(* IEC 61131-3 sources: Swiity/AutomationStudio/VendingMachine, 4 files *)

(* ---- Types.typ ---- *)
(*
  Types.typ
  Vending Machine Project – User-Defined Data Types (UDT)
  IEC 61131-3 Structured Text  |  B&R Automation Studio
*)

TYPE
  (* ---------------------------------------------------------------
     State enumeration for the main vending-machine state machine
  --------------------------------------------------------------- *)
  VendingState_e : (
    STATE_IDLE         := 0,   (* Waiting for coin / card input        *)
    STATE_COIN_CHECK   := 1,   (* Validating inserted coin             *)
    STATE_SELECT       := 2,   (* Product selection active             *)
    STATE_DISPENSE     := 3,   (* Dispensing selected product          *)
    STATE_COLLECT      := 4,   (* Waiting for customer to collect      *)
    STATE_CHANGE       := 5,   (* Returning change                     *)
    STATE_ERROR        := 6,   (* Error / fault state                  *)
    STATE_MAINTENANCE  := 7    (* Maintenance / refill mode            *)
  );

  (* ---------------------------------------------------------------
     Product slot descriptor
  --------------------------------------------------------------- *)
  ProductSlot_t : STRUCT
    Name        : STRING[32];  (* Product name                         *)
    Price       : REAL;        (* Price in the local currency unit     *)
    Quantity    : UINT;        (* Remaining stock count                *)
    SlotActive  : BOOL;        (* TRUE = slot is enabled               *)
  END_STRUCT;

  (* ---------------------------------------------------------------
     Coin / payment input data
  --------------------------------------------------------------- *)
  PaymentData_t : STRUCT
    CoinInserted    : BOOL;    (* Coin-drop sensor signal              *)
    CoinValue       : REAL;    (* Value detected by coin validator     *)
    TotalCredit     : REAL;    (* Accumulated credit                   *)
    CreditAccepted  : BOOL;    (* Sufficient credit for selection      *)
  END_STRUCT;

  (* ---------------------------------------------------------------
     Sensor input bundle (mapped from Arduino via serial / I/O)
  --------------------------------------------------------------- *)
  SensorInputs_t : STRUCT
    CoinSensor       : BOOL;   (* Coin-drop detection                  *)
    ProductSensor    : BOOL;   (* Product dispensed / collected        *)
    TempSensor       : REAL;   (* Cabinet temperature (°C)             *)
    DoorSensor       : BOOL;   (* Service door open                    *)
    StockSensor      : ARRAY[0..7] OF BOOL; (* Per-slot stock presence *)
  END_STRUCT;

  (* ---------------------------------------------------------------
     Actuator output bundle (mapped to Arduino via serial / I/O)
  --------------------------------------------------------------- *)
  ActuatorOutputs_t : STRUCT
    MotorEnable      : BOOL;              (* Dispense motor enable      *)
    MotorSlot        : UINT;              (* Target slot index          *)
    ChangeMechanism  : BOOL;              (* Activate change dispenser  *)
    DisplayMsg       : STRING[64];        (* LCD / display message      *)
    StatusLED        : BOOL;              (* Status indicator LED       *)
    CoolingFan       : BOOL;              (* Cooling fan control        *)
  END_STRUCT;

END_TYPE

(* ---- Variables.var ---- *)
(*
  Variables.var
  Vending Machine Project – Global Variable Declarations
  IEC 61131-3 Structured Text  |  B&R Automation Studio
*)

VAR_GLOBAL

  (* ---------------------------------------------------------------
     State machine
  --------------------------------------------------------------- *)
  gState          : VendingState_e := STATE_IDLE;
  gPrevState      : VendingState_e := STATE_IDLE;

  (* ---------------------------------------------------------------
     Product configuration  (8 slots, indices 0..7)
  --------------------------------------------------------------- *)
  gProductSlots   : ARRAY[0..7] OF ProductSlot_t;
  gSelectedSlot   : UINT := 0;

  (* ---------------------------------------------------------------
     Payment
  --------------------------------------------------------------- *)
  gPayment        : PaymentData_t;

  (* ---------------------------------------------------------------
     I/O bundles (exchanged with Arduino via serial / fieldbus)
  --------------------------------------------------------------- *)
  gSensors        : SensorInputs_t;
  gActuators      : ActuatorOutputs_t;

  (* ---------------------------------------------------------------
     Timing
  --------------------------------------------------------------- *)
  gDispenseTimer  : TON;         (* Motor run time-out                 *)
  gCollectTimer   : TON;         (* Collect reminder time-out          *)
  gErrorTimer     : TON;         (* Error-reset delay                  *)

  (* ---------------------------------------------------------------
     Diagnostics / HMI
  --------------------------------------------------------------- *)
  gErrorCode      : UINT  := 0;
  gTotalSales     : UDINT := 0;  (* Number of successful vend cycles   *)
  gHmiMessage     : STRING[64];

END_VAR

VAR_GLOBAL CONSTANT

  (* ---------------------------------------------------------------
     Application constants
  --------------------------------------------------------------- *)
  cNumSlots           : UINT := 8;        (* Total number of product slots    *)
  cDispenseTimeMs     : TIME := T#3000ms; (* Motor run duration               *)
  cCollectTimeoutMs   : TIME := T#30000ms;(* Collect reminder after 30 s      *)
  cMinTemperature     : REAL := 2.0;      (* Min cabinet temperature (°C)     *)
  cMaxTemperature     : REAL := 10.0;     (* Max cabinet temperature (°C)     *)

END_VAR

(* ---- StateMachine.st ---- *)
(*
  StateMachine.st
  Vending Machine Project – State-Machine Logic
  IEC 61131-3 Structured Text  |  B&R Automation Studio

  Call this function block once per PLC cycle from Main.st.
*)

FUNCTION_BLOCK VendingStateMachine

VAR_INPUT
  Sensors   : SensorInputs_t;   (* Live sensor data                    *)
END_VAR

VAR_OUTPUT
  Actuators : ActuatorOutputs_t;(* Computed actuator commands          *)
  State     : VendingState_e;   (* Current state (for HMI / logging)   *)
END_VAR

VAR
  _dispenseTimer   : TON;
  _collectTimer    : TON;
  _errorTimer      : TON;
  _coinSensorPrev  : BOOL := FALSE; (* Previous coin-sensor state for edge detection *)
END_VAR

(* ---------------------------------------------------------------
   Main state-machine CASE statement
--------------------------------------------------------------- *)
CASE gState OF

  (* ---- IDLE -------------------------------------------------- *)
  STATE_IDLE:
    Actuators.DisplayMsg  := 'Insert coin';
    Actuators.StatusLED   := TRUE;
    Actuators.MotorEnable := FALSE;

    IF Sensors.CoinSensor THEN
      gState := STATE_COIN_CHECK;
    END_IF

  (* ---- COIN CHECK -------------------------------------------- *)
  STATE_COIN_CHECK:
    Actuators.DisplayMsg := 'Checking coin...';

    (* Accumulate credit on rising edge of coin sensor only *)
    IF Sensors.CoinSensor AND NOT _coinSensorPrev THEN
      gPayment.TotalCredit := gPayment.TotalCredit + gPayment.CoinValue;
    END_IF
    _coinSensorPrev := Sensors.CoinSensor;

    (* Always allow product selection once any credit exists *)
    IF gPayment.TotalCredit > 0.0 THEN
      gState := STATE_SELECT;
    END_IF

  (* ---- SELECT ------------------------------------------------ *)
  STATE_SELECT:
    Actuators.DisplayMsg := 'Select product (0-7)';

    (* Validate selection: slot must be active and affordable *)
    IF gSelectedSlot < cNumSlots
       AND gProductSlots[gSelectedSlot].SlotActive
       AND gProductSlots[gSelectedSlot].Quantity > 0
       AND gPayment.TotalCredit >= gProductSlots[gSelectedSlot].Price THEN

      gPayment.CreditAccepted := TRUE;
      gState := STATE_DISPENSE;
    END_IF

  (* ---- DISPENSE ---------------------------------------------- *)
  STATE_DISPENSE:
    Actuators.DisplayMsg      := 'Dispensing...';
    Actuators.MotorEnable     := TRUE;
    Actuators.MotorSlot       := gSelectedSlot;

    _dispenseTimer(IN := TRUE, PT := cDispenseTimeMs);

    IF _dispenseTimer.Q THEN
      _dispenseTimer(IN := FALSE);
      Actuators.MotorEnable := FALSE;

      (* Deduct price, update stock *)
      gPayment.TotalCredit                       := gPayment.TotalCredit
                                                    - gProductSlots[gSelectedSlot].Price;
      gProductSlots[gSelectedSlot].Quantity      := gProductSlots[gSelectedSlot].Quantity - 1;
      gTotalSales                                := gTotalSales + 1;

      gState := STATE_COLLECT;
    END_IF

  (* ---- COLLECT ----------------------------------------------- *)
  STATE_COLLECT:
    Actuators.DisplayMsg := 'Please collect your item';
    _collectTimer(IN := TRUE, PT := cCollectTimeoutMs);

    IF Sensors.ProductSensor OR _collectTimer.Q THEN
      _collectTimer(IN := FALSE);
      gState := STATE_CHANGE;
    END_IF

  (* ---- CHANGE ----------------------------------------------- *)
  STATE_CHANGE:
    IF gPayment.TotalCredit > 0.0 THEN
      Actuators.DisplayMsg     := 'Returning change';
      Actuators.ChangeMechanism := TRUE;
    ELSE
      Actuators.ChangeMechanism := FALSE;
      gPayment.TotalCredit      := 0.0;
      gPayment.CreditAccepted   := FALSE;
      gState := STATE_IDLE;
    END_IF

    (* Once credit is cleared, return to idle *)
    IF gPayment.TotalCredit <= 0.0 THEN
      Actuators.ChangeMechanism := FALSE;
      gState := STATE_IDLE;
    END_IF

  (* ---- ERROR ------------------------------------------------- *)
  STATE_ERROR:
    Actuators.DisplayMsg  := 'Error – call service';
    Actuators.StatusLED   := NOT Actuators.StatusLED; (* Blink *)
    Actuators.MotorEnable := FALSE;

    _errorTimer(IN := TRUE, PT := T#5000ms);
    IF _errorTimer.Q THEN
      _errorTimer(IN := FALSE);
      gErrorCode := 0;
      gState     := STATE_IDLE;
    END_IF

  (* ---- MAINTENANCE ------------------------------------------ *)
  STATE_MAINTENANCE:
    Actuators.DisplayMsg := 'Maintenance mode';
    Actuators.StatusLED  := FALSE;
    (* Maintenance logic handled by HMI / operator *)

  ELSE
    gState := STATE_ERROR;

END_CASE

(* ---------------------------------------------------------------
   Temperature monitoring (runs in every state)
--------------------------------------------------------------- *)
IF Sensors.TempSensor > cMaxTemperature THEN
  Actuators.CoolingFan := TRUE;
ELSIF Sensors.TempSensor < cMinTemperature THEN
  Actuators.CoolingFan := FALSE;
END_IF

(* ---------------------------------------------------------------
   Service door interlock
--------------------------------------------------------------- *)
IF Sensors.DoorSensor AND gState <> STATE_MAINTENANCE THEN
  gState              := STATE_MAINTENANCE;
  Actuators.MotorEnable := FALSE;
END_IF

State     := gState;

END_FUNCTION_BLOCK

(* ---- Main.st ---- *)
(*
  Main.st
  Vending Machine Project – Main Cyclic Task
  IEC 61131-3 Structured Text  |  B&R Automation Studio

  This program is called once per PLC scan cycle.
  It wires the state-machine function block to global I/O variables.
*)

PROGRAM MAIN

VAR
  fbVending : VendingStateMachine; (* State-machine function block instance *)
END_VAR

(* ---------------------------------------------------------------
   Call the vending state machine every cycle
--------------------------------------------------------------- *)
fbVending(
  Sensors   := gSensors,
  Actuators => gActuators,
  State     => gState
);

(* ---------------------------------------------------------------
   Mirror outputs to HMI display string
--------------------------------------------------------------- *)
gHmiMessage := gActuators.DisplayMsg;

END_PROGRAM
